(* PLC project relay, Dassault Systèmes ControlBuild 2024x *)
(* stored: creationDateTime 2023-10-03T11:13:23-01:00 *)

(* This module simulates a relay or a contactor with its auxiliary contact. *)
FUNCTION_BLOCK equipment_library.relay
  VAR_INPUT
    contactorInterlock : BOOL := false;
    cmdSupply : BOOL := true;
    sensorSupply : BOOL := true;
    energyBefore : BOOL := true;
  END_VAR
  VAR_OUTPUT
    interlockFB : BOOL := false;
    energyAfter : BOOL := false;
  END_VAR
  VAR
    memoInterlock : BOOL := false;
  END_VAR
  VAR CONSTANT
    interlockLogic : BOOL := true;
  END_VAR
  VAR
    d_interlock : BOOL := false;
    v_d_interlock : BOOL := true;
  END_VAR


ACTION C_source_code:
/* ----------------------------------------------------------------	*/
/* Type : Model of Operative Behaviour					*/
/* Category :  Power								*/
/* Author : Dassault Systemes						*/
/* Update date : June 2010							*/
/* ----------------------------------------------------------------	*/
/* This module simulates a relay or a contactor 			*/
/* 	with its auxiliary contact.						*/
/* ----------------------------------------------------------------	*/

/* ----------------------------------------------------------------	*/
/* Management of orders from Control Part					*/
/*	if there is no power supply for command 				*/
/*         the contactor doesn't understand the control order		*/
/*     Fault is mechanical fault.						*/
/* ----------------------------------------------------------------	*/
if (d_interlock) interlockFB=v_d_interlock;
else memoInterlock=contactorInterlock && cmdSupply;

/* ----------------------------------------------------------------	*/
/* Calculation of the on-state of energy					*/
/* If there is no energy downstream there is no energy downstream	*/
/* ----------------------------------------------------------------	*/
energyAfter=memoInterlock & energyBefore;

/* ----------------------------------------------------------------	*/
/* Management of feedback to Control Part					*/
/*	if there is no power supply for the sensor			*/
/*         there is no contactor feedback.				*/
/*     else contactor feedback returns its state combined with	*/
/*	    wiring logic (its default value is : positive).		*/
/* ----------------------------------------------------------------	*/
interlockFB=(memoInterlock ^ !interlockLogic) && sensorSupply;
END_ACTION
END_FUNCTION_BLOCK
